FUNCTION_BLOCK PUBLIC PAEdge EXTENDS ACObject IMPLEMENTS IACEdge
VAR_INPUT
END_VAR
VAR_OUTPUT
END_VAR
VAR
	_Source : IACPoint;	
	_Target : IACPoint;	
	_ConnectionType : ConnectionTypesEnum;	
	
	// Gibt an, dass dieser Weg gerade von einer Funktion verwendet wird
	_AllocatedByFunction : IPAProcessFunction;
END_VAR

PROPERTY ACUrlS : STRING
GET
VAR
	str : STRING(200);
END_VAR
str := CONCAT(Source.ACUrlS, + '|');
str := CONCAT(str, + Target.ACUrlS);
ACUrlS := str;
END_GET
END_PROPERTY

PROPERTY AllocatedByFunction : IPAProcessFunction
GET
AllocatedByFunction := _AllocatedByFunction;
END_GET
SET
_AllocatedByFunction := AllocatedByFunction;
END_SET
END_PROPERTY

// Compares if ACUrl of Source and Target are identical
METHOD Compare : BOOL
VAR_INPUT
	edge : IACEdge;	
END_VAR
VAR
	// Explizite Deklaration notwendig, weil Properties nicht verglichen werden können :-(
	sourceP1 : IACPoint;
	targetP1 : IACPoint;
	sourceC1 : IACComponent;
	targetC1 : IACComponent;
	sourceP2 : IACPoint;
	targetP2 : IACPoint;
	sourceC2 : IACComponent;
	targetC2 : IACComponent;
END_VAR
IF edge = 0 THEN
	Compare := FALSE;
	RETURN;
END_IF

sourceP1 := Source;
targetP1 := Target;
IF 	   sourceP1 = 0 OR targetP1 = 0 THEN
	Compare := FALSE;
	RETURN;	
END_IF

sourceP2 := edge.Source;
targetP2 := edge.Target;
IF 	   sourceP2 = 0 OR targetP2 = 0 THEN
	Compare := FALSE;
	RETURN;	
END_IF


sourceC1 := sourceP1.Parent;
targetC1 := targetP1.Parent;
IF 	   sourceC1 = 0 OR targetC1 = 0 THEN
	Compare := FALSE;
	RETURN;	
END_IF

sourceC2 := sourceP2.Parent;
targetC2 := targetP2.Parent;
IF 	   sourceC2 = 0 OR targetC2 = 0 THEN
	Compare := FALSE;
	RETURN;	
END_IF

IF (sourceC1.ACUrl = sourceC2.ACUrl AND targetC1.ACUrl = targetC2.ACUrl) THEN
	Compare := TRUE;
	RETURN;			
END_IF

Compare := FALSE;
END_METHOD

PROPERTY ConnectionType : ConnectionTypesEnum
GET
ConnectionType := _ConnectionType;
END_GET
END_PROPERTY

METHOD FB_init : BOOL
VAR_INPUT
	bInitRetains : BOOL; // if TRUE, the retain variables are initialized (warm start / cold start)
	bInCopyCode : BOOL;  // if TRUE, the instance afterwards gets moved into the copy code (online change)
	source : IACPoint;
	target : IACPoint;
	connectionType : ConnectionTypesEnum;
END_VAR

VAR
	isValidRef: BOOL;
END_VAR
IF source <> 0 AND target <> 0 THEN
	_Source := source;
	_Target := target;
END_IF
_ConnectionType := connectionType;
IncFBInitCount();
END_METHOD

METHOD FB_postinit
VAR_INPUT
		root : IACVariobatch;
END_VAR
SUPER^.FB_postinit(root);
END_METHOD

PROPERTY Source : IACPoint
GET
Source := _Source;
END_GET
END_PROPERTY

PROPERTY Target : IACPoint
GET
Target := _Target;
END_GET
END_PROPERTY

PROPERTY TypeOfACObject : TypeOfACObjectEnum
GET
TypeOfACObject := TypeOfACObjectEnum.Edge;
END_GET
END_PROPERTY

END_FUNCTION_BLOCK

(* stored: Version 1.1.0.1, ProductVersion 3.1.4022.7
   POU PAEdge: Id {b1628018-e515-4bd3-bf50-33e399f22b02}, SpecialFunc None
   Property ACUrlS: Id {13194f77-f58f-4414-82df-f2ea33e2a4aa}
   Get Get: Id {b38d25c4-a4ac-47d4-8bf9-6538682f1938}
   Property AllocatedByFunction: Id {436ab8e0-6a7e-4a19-b2be-b5fa77f7f2f8}
   Get Get: Id {f8b8b2ed-c789-477b-8390-eaff26fdf05e}
   Set Set: Id {2e0760ab-18bf-48f1-bafe-541c4dbd38ef}
   Method Compare: Id {1c7455bb-39d7-42dd-89e4-8cb9d9f0fa09}
   Property ConnectionType: Id {bb87e033-ce4f-4de4-9bcd-20215dc5ec3d}
   Get Get: Id {e1f1277b-7e1c-43cf-88ef-1a4d0f6ec209}
   Method FB_init: Id {969e98d1-950b-4913-b198-648678ef9fc0}
   Method FB_postinit: Id {ace20de9-c8e2-4a93-af46-712625169229}
   Property Source: Id {dec7f72d-15f2-4d11-b348-e24e0be90e83}
   Get Get: Id {7c2ae090-5470-440c-8376-8c790a0efa4b}
   Property Target: Id {fc0d937b-58c0-49fc-ab35-2f33d352117f}
   Get Get: Id {75dbb33a-9784-4b32-9035-f68bdafbf2f8}
   Property TypeOfACObject: Id {c631f490-5f1c-45a4-994d-18fa8461cba4}
   Get Get: Id {eb3604fd-5b22-4a7d-ac18-a618296d5340} *)
